FUNCTION_BLOCK SCOPE
  (* Standard: 61499-2 *)
  (* Version 03-07-12, GASR *)
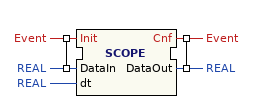
  EVENT_INPUT
    Init WITH DataIn;
  END_EVENT
  EVENT_OUTPUT
    Cnf WITH DataOut;
  END_EVENT
  VAR_INPUT
    DataIn : REAL;
    dt : REAL;
  END_VAR
  VAR_OUTPUT
    DataOut : REAL;
  END_VAR
  SERVICE SCOPE/User
    SEQUENCE Scope
      SCOPE.Init() -> User.Cnf();
      User.Done() -> SCOPE.cnf();
    END_SEQUENCE
  END_SERVICE
END_FUNCTION_BLOCK
